// TwinCAT 3 PLC project sortingbyheight
// ProgramVersion: 3.1.4024.12
// libraries:
//   Tc2_ModbusSrv, * (Beckhoff Automation GmbH)
//   Tc2_Standard, * (Beckhoff Automation GmbH)
//   Tc2_System, * (Beckhoff Automation GmbH)
//   Tc3_Module, * (Beckhoff Automation GmbH)
//   Util, * (System)
// project tree:
//   GVLs/ GeneralTags.TcGVL, GVL.TcGVL, IO.TcGVL
//   / PlcTask.TcTTO
//   POUs/Comms/ InputOutput.TcPOU, Modbus_ReadInputs.TcPOU, Modbus_WriteOutputs.TcPOU
//   POUs/Main/ MAIN.TcPOU
//   POUs/System/ ConveyorEntry.TcPOU, ElectricBoard.TcPOU, System.TcPOU, TransferConveyor.TcPOU, TransferToLeftorRight.TcPOU
// real-time tasks:
//   TASK PlcTask: cycle T#10ms, priority 20, ADS port 350

CONFIGURATION sortingbyheight
    RESOURCE PLC ON TwinCAT3
        TASK PlcTask(INTERVAL := T#10ms, PRIORITY := 20);
        PROGRAM MAIN WITH PlcTask : MAIN;
    END_RESOURCE
END_CONFIGURATION

// ---- GVLs/GeneralTags.TcGVL
VAR_GLOBAL
	SystemStarted		: BOOL;
	FlashBit			: BOOL;
	TransferBusy		: BOOL;
	TransferringLeft	: BOOL;
	TransferringRight	: BOOL;
	EmergencyActivated	: BOOL;
	BoxCounted			: WORD;
END_VAR

// ---- GVLs/GVL.TcGVL
VAR_GLOBAL
	InputArea	: ARRAY[0..15] OF BYTE;
	OutputArea	: ARRAY[0..15] OF BYTE;
END_VAR

// ---- GVLs/IO.TcGVL
VAR_GLOBAL
	//Inputs
	High_Sensor 	:	BOOL;
	Low_Sensor 		:	BOOL;
	Pallet_Sensor 	:	BOOL;
	Loaded			:	BOOL;
	At_Left_Entry	:	BOOL;
	At_Left_Exit	:	BOOL;
	At_Right_Entry	:	BOOL;
	At_Right_Exit	:	BOOL;
	Start			:	BOOL;
	Reset			:	BOOL;
	Stop			:	BOOL;
	Emergency_Stop	:	BOOL;
	Auto			:	BOOL;
	FactoryIO_RUN	:	BOOL;
	//Outputs
	Conveyor_Entry	:	BOOL;
	Load			:	BOOL;
	Unload			:	BOOL;
	Transfer_Left	: 	BOOL;
	Transfer_Right	: 	BOOL;
	Conveyor_Left	: 	BOOL;
	Conveyor_Right	: 	BOOL;
	Start_Light		:	BOOL;
	Reset_Light		:	BOOL;
	Stop_Light		:	BOOL;
END_VAR

// ---- POUs/Main/MAIN.TcPOU
PROGRAM MAIN
VAR
	Flash: BLINK;
END_VAR

//Comms
Modbus_ReadInputs();
Modbus_WriteOutputs();
InputOutput();

//System
System();
Flash(ENABLE:= TRUE , TIMELOW:= T#500MS, TIMEHIGH:= T#500MS, OUT=> FlashBit);

END_PROGRAM

// ---- POUs/Comms/Modbus_ReadInputs.TcPOU
PROGRAM Modbus_ReadInputs
VAR
	bReadInputs : 	BOOL;
	tReadInputs	: 	TON;
	ReadInputs	: FB_MBReadInputs;

END_VAR

//Modbus read inputs function.
tReadInputs(IN:= NOT ReadInputs.bBusy, PT:= T#10MS , Q=> bReadInputs, ET=> );

ReadInputs(
	sIPAddr:= '127.0.0.1', 
	nTCPPort:= 505, 
	nUnitID:= 255, 
	nQuantity:= 14, 
	nMBAddr:= 0, 
	cbLength:= SIZEOF(InputArea), 
	pDestAddr:= ADR(InputArea), 
	bExecute:= bReadInputs, 
	tTimeout:= T#1S, 
	bBusy=> , 
	bError=> , 
	nErrId=> , 
	cbRead=> );

END_PROGRAM

// ---- POUs/Comms/Modbus_WriteOutputs.TcPOU
PROGRAM Modbus_WriteOutputs
VAR
	bWriteOutput: BOOL;
	tWriteOutput: TON;
	WriteOutputs: FB_MBWriteCoils;

	ModbusWriteSingle: FB_MBWriteSingleReg;
	ModbusSingleWrite: TON;
	bWriteSingleReg: BOOL;
END_VAR

//Modbus write outputs function.
tWriteOutput(IN:= NOT WriteOutputs.bBusy , PT:= T#10MS, Q=> bWriteOutput , ET=> );

WriteOutputs(
	sIPAddr:= '127.0.0.1', 
	nTCPPort:= 505, 
	nUnitID:= 255, 
	nQuantity:= 10, 
	nMBAddr:= 0, 
	cbLength:= SIZEOF(OutputArea), 
	pSrcAddr:= ADR(OutputArea), 
	bExecute:= bWriteOutput, 
	tTimeout:= T#1S, 
	bBusy=> , 
	bError=> , 
	nErrId=> );

ModbusSingleWrite(IN:= NOT ModbusWriteSingle.bBusy, PT:=T#10MS , Q=> bWriteSingleReg, ET=> );
	
ModbusWriteSingle(
	sIPAddr:= '127.0.0.1', 
	nTCPPort:= 505, 
	nUnitID:= 255, 
	nMBAddr:= 0, 
	nValue:= BoxCounted, 
	bExecute:= bWriteSingleReg, 
	tTimeout:= T#1S, 
	bBusy=> , 
	bError=> , 
	nErrId=> );

END_PROGRAM

// ---- POUs/Comms/InputOutput.TcPOU
PROGRAM InputOutput
VAR
END_VAR

//Inputs
High_Sensor 	:= InputArea[0].0;
Low_Sensor 		:= InputArea[0].1;
Pallet_Sensor 	:= InputArea[0].2;
Loaded			:= InputArea[0].3;
At_Left_Entry	:= InputArea[0].4;
At_Left_Exit	:= InputArea[0].5;
At_Right_Entry	:= InputArea[0].6;
At_Right_Exit	:= InputArea[0].7;
Start			:= InputArea[1].0;
Reset			:= InputArea[1].1;
Stop			:= InputArea[1].2;
Emergency_Stop	:= InputArea[1].3;
Auto			:= InputArea[1].4;
FactoryIO_RUN	:= InputArea[1].5;
//Outputs
OutputArea[0].0	:= Conveyor_Entry;
OutputArea[0].1 := Load;
OutputArea[0].2 := Unload;
OutputArea[0].3 := Transfer_Left;
OutputArea[0].4 := Transfer_Right;
OutputArea[0].5 := Conveyor_Left;
OutputArea[0].6 := Conveyor_Right;
OutputArea[0].7 := Start_Light;
OutputArea[1].0 := Reset_Light;
OutputArea[1].1 := Stop_Light;
//If emergency stop is activated, reset all outputs and system memory bits to zero. 
IF EmergencyActivated THEN
	Conveyor_Entry		:= 0;
	Load 				:= 0;
	Unload 				:= 0;
	Transfer_Left 		:= 0;
	Transfer_Right 		:= 0;
	Conveyor_Left 		:= 0;
	Conveyor_Right 		:= 0;
	Start_Light 		:= 0;
	Stop_Light 			:= 0;
	SystemStarted		:= FALSE;
	TransferBusy		:= FALSE;
	TransferringLeft	:= FALSE;
	TransferringRight	:= FALSE;
END_IF

END_PROGRAM

// ---- POUs/System/System.TcPOU
PROGRAM System
VAR
	ElectricBoard: ElectricBoard;
	ConveyorEntry: ConveyorEntry;
	TransferConveyor: TransferConveyor;
	TransferToLeftorRight: TransferToLeftorRight;
END_VAR

//System functions.
ElectricBoard();
ConveyorEntry();
TransferConveyor();
TransferToLeftorRight();

END_PROGRAM

// ---- POUs/System/ElectricBoard.TcPOU
FUNCTION_BLOCK ElectricBoard
VAR_INPUT
END_VAR
VAR_OUTPUT
END_VAR
VAR
	EmergencyBlock: SR;
END_VAR

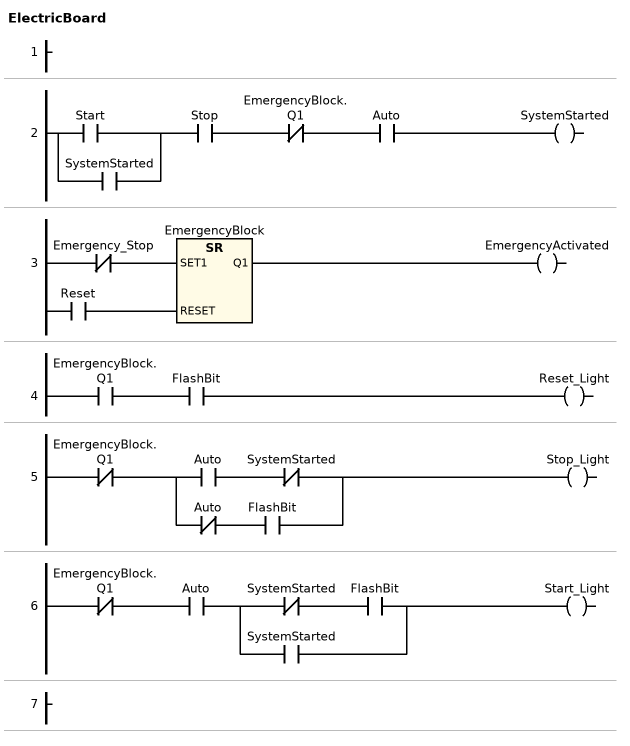
// NETWORK 1

// NETWORK 2
SystemStarted := (Start OR SystemStarted) AND Stop AND NOT EmergencyBlock.Q1 AND Auto;

// NETWORK 3
EmergencyBlock(SET1 := NOT Emergency_Stop, RESET := Reset); // SR
EmergencyActivated := EmergencyBlock.Q1;

// NETWORK 4
Reset_Light := EmergencyBlock.Q1 AND FlashBit;

// NETWORK 5
Stop_Light := NOT EmergencyBlock.Q1 AND (Auto AND NOT SystemStarted OR NOT Auto AND FlashBit);

// NETWORK 6
Start_Light := NOT EmergencyBlock.Q1 AND Auto AND (NOT SystemStarted AND FlashBit OR SystemStarted);

// NETWORK 7

END_FUNCTION_BLOCK

// ---- POUs/System/ConveyorEntry.TcPOU
FUNCTION_BLOCK ConveyorEntry
VAR_INPUT
END_VAR
VAR_OUTPUT
END_VAR
VAR
	ConveyorEntryToken : INT;
END_VAR

//If emergency button is activated or system isn't started or stopped, reset system token to 10.
IF NOT SystemStarted OR EmergencyActivated THEN
	ConveyorEntryToken := 10;
END_IF
//Conveyor entry system conditions.
CASE ConveyorEntryToken OF
	//
	10:
		//Waiting for system start
		IF SystemStarted THEN
			ConveyorEntryToken := 20;
		END_IF
	20:
		//Start conveyor entry motor when system is started. Continue to work until pallet is loaded or if loaded already , work until pallet sensor activates.
		Conveyor_Entry := TRUE;
		IF TransferBusy AND Pallet_Sensor THEN
			ConveyorEntryToken := 30;
		ELSIF NOT TransferBusy AND Loaded THEN
			ConveyorEntryToken := 30;
		END_IF
	30:
		//Stop until pallet is pushed one side completely. 
		Conveyor_Entry := FALSE;
		IF NOT TransferBusy AND NOT Loaded THEN
			ConveyorEntryToken := 20;
		END_IF
ELSE
	ConveyorEntryToken := 10;
END_CASE

END_FUNCTION_BLOCK

// ---- POUs/System/TransferConveyor.TcPOU
FUNCTION_BLOCK TransferConveyor
VAR_INPUT
END_VAR
VAR_OUTPUT
END_VAR
VAR
	TransferConveyorToken : INT;
	PalletSensorNegEdge: F_TRIG;
	LeftEntryPosEdge: R_TRIG;
	RightEntryPosEdge: R_TRIG;
	
	PalletNegative : BOOL;
	LeftEntryPositive : BOOL;
	RightEntryPositive : BOOL;	


END_VAR

//If emergency button is activated or system isn't started or stopped, reset system token to 10.
IF NOT SystemStarted OR EmergencyActivated THEN
	TransferConveyorToken := 10;
END_IF
//Positive or negative edges of sensors.
PalletSensorNegEdge(CLK:= Pallet_Sensor, Q=> PalletNegative );
LeftEntryPosEdge(CLK:= At_Left_Entry , Q=> LeftEntryPositive );
RightEntryPosEdge(CLK:= At_Right_Entry , Q=> RightEntryPositive );
//Transfer conveyors working conditions.
CASE TransferConveyorToken OF
	//
	10:
		//Waiting for system start
		IF SystemStarted THEN
			TransferConveyorToken := 20;
		ELSE
			Transfer_Left := FALSE;
			Transfer_Right := FALSE;
		END_IF
	20:
		//Reset everything and wait for a new pallet.
		Load := FALSE;
		Transfer_Left := FALSE;
		Transfer_Right := FALSE;
		TransferringLeft := FALSE;
		TransferringRight := FALSE;
		
		IF Pallet_Sensor THEN
			TransferConveyorToken := 30;
		END_IF
	30:
		//Start loading conveyor until loaded sensor is activated. And decide where to transfer pallet according to low and high sensors.
		Load := TRUE;
		//
		IF Pallet_Sensor AND Low_Sensor AND NOT High_Sensor THEN
			TransferringLeft := TRUE;
		ELSIF Pallet_Sensor AND Low_Sensor AND High_Sensor THEN
			TransferringRight := TRUE;
		ELSIF PalletNegative THEN
			TransferBusy := TRUE;
		ELSIF Loaded AND TransferringLeft THEN
			TransferConveyorToken := 40;
		ELSIF Loaded AND TransferringRight THEN
			TransferConveyorToken := 50;
		END_IF
	
	40:
		//If the box is small, transfer it to left.
		Load := FALSE;
		Transfer_Left := TRUE;
		
		IF LeftEntryPositive THEN
			TransferBusy := FALSE;
			TransferConveyorToken := 10;
		END_IF
	
		
	50:
		//If the box is high, transfer it to right.
		Load := FALSE;
		Transfer_Right := TRUE;
		
		IF RightEntryPositive THEN
			TransferBusy := FALSE;
			TransferConveyorToken := 10;
		END_IF	
		
	ELSE
		//
		TransferConveyorToken := 10;
END_CASE

END_FUNCTION_BLOCK

// ---- POUs/System/TransferToLeftorRight.TcPOU
FUNCTION_BLOCK TransferToLeftorRight
VAR_INPUT
END_VAR
VAR_OUTPUT
END_VAR
VAR
	LeftExitPosEdge: R_TRIG;
	LeftExitPositive: BOOL;
	RightExitPosEdge: R_TRIG;
	RightExitPositive: BOOL;
	LeftConveyorCounter: CTUD;
	RightConveyorCounter: CTUD;
	BoxCounter: CTU;
END_VAR


//Positive edges of the sensors.
LeftExitPosEdge(CLK:= At_Left_Exit, Q=> LeftExitPositive );
RightExitPosEdge(CLK:= At_Right_Exit, Q=> RightExitPositive);
//Left conveyor box counter.
LeftConveyorCounter(
	CU:= NOT At_Left_Entry , 
	CD:= LeftExitPositive, 
	RESET:= EmergencyActivated, 
	LOAD:= , 
	PV:= , 
	QU=> , 
	QD=> , 
	CV=> );
//Right conveyor box counter.	
RightConveyorCounter(
	CU:= NOT At_Right_Entry, 
	CD:= RightExitPositive, 
	RESET:= EmergencyActivated, 
	LOAD:= , 
	PV:= , 
	QU=> , 
	QD=> , 
	CV=> );
//Left conveyor works until it is empty.
IF NOT LeftConveyorCounter.QD THEN
	Conveyor_Left := TRUE;
ELSE
	Conveyor_Left := FALSE;
END_IF
//Right conveyor works until it is empty.
IF NOT RightConveyorCounter.QD THEN
	Conveyor_Right := TRUE;
ELSE
	Conveyor_Right := FALSE;
END_IF
//Total box counter.
BoxCounter(
	CU:= LeftExitPositive OR RightExitPositive, 
	RESET:= EmergencyActivated, 
	PV:= , 
	Q=> , 
	CV=> );

BoxCounted := BoxCounter.CV;

END_FUNCTION_BLOCK
